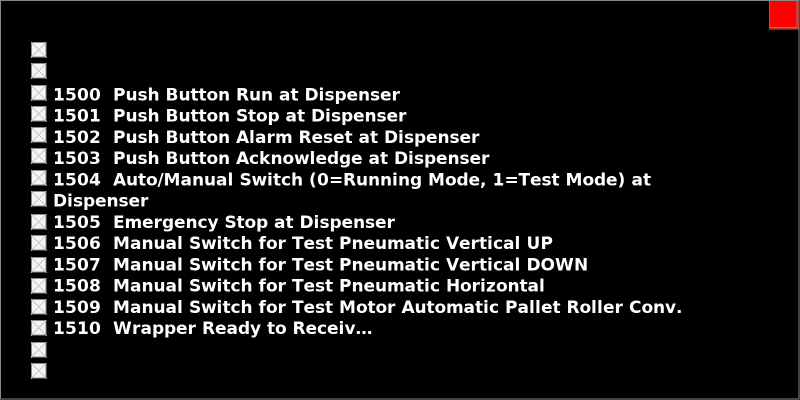
VISUALIZATION P2_DI6  // 800x400, background image 
    ImageSwitcher (31,42 15x15), variable: InputOutput_GVL.Digital_Input[81], behaviour: TOGGLE
    Label (50,16 677x391), "1500 Push Button Run at Dispenser 1501 Push Button Stop at Dispenser 1502 Push Button Alarm Reset at Dispenser 1503 Push Button Acknowledge at Dispenser 1504 Auto/Manual Switch (0=Running Mode, 1=Test Mode) at Dispenser 1505 Emergency Stop at Dispenser 1506 Manual Switch for Test Pneumatic Vertical UP 1507 Manual Switch for Test Pneumatic Vertical DOWN 1508 Manual Switch for Test Pneumatic Horizontal 1509 Manual Switch for Test Motor Automatic Pallet Roller Conv. 1510 Wrapper Ready to Receive 1511 End of Transfer Pallet in Infeed 1512 Pallet Ready in Outfeed 1513 Emergency Stop Wrapper is Active 1514 Status Bypass Wrapper Existing 1515 Pressure Switch for Pallet Dispenser"
    ImageSwitcher (31,63 15x15), variable: InputOutput_GVL.Digital_Input[82], behaviour: TOGGLE
    ImageSwitcher (31,85 15x15), variable: InputOutput_GVL.Digital_Input[83], behaviour: TOGGLE
    ImageSwitcher (31,106 15x15), variable: InputOutput_GVL.Digital_Input[84], behaviour: TOGGLE
    ImageSwitcher (31,127 15x15), variable: InputOutput_GVL.Digital_Input[85], behaviour: TOGGLE
    ImageSwitcher (31,148 15x15), variable: InputOutput_GVL.Digital_Input[86], behaviour: TOGGLE
    ImageSwitcher (31,170 15x15), variable: InputOutput_GVL.Digital_Input[87], behaviour: TOGGLE
    ImageSwitcher (31,191 15x15), variable: InputOutput_GVL.Digital_Input[88], behaviour: TOGGLE
    ImageSwitcher (31,214 15x15), variable: InputOutput_GVL.Digital_Input[89], behaviour: TOGGLE
    ImageSwitcher (31,235 15x15), variable: InputOutput_GVL.Digital_Input[90], behaviour: TOGGLE
    ImageSwitcher (31,257 15x15), variable: InputOutput_GVL.Digital_Input[91], behaviour: TOGGLE
    ImageSwitcher (31,278 15x15), variable: InputOutput_GVL.Digital_Input[92], behaviour: TOGGLE
    ImageSwitcher (31,299 15x15), variable: InputOutput_GVL.Digital_Input[93], behaviour: TOGGLE
    ImageSwitcher (31,320 15x15), variable: InputOutput_GVL.Digital_Input[94], behaviour: TOGGLE
    ImageSwitcher (31,342 15x15), variable: InputOutput_GVL.Digital_Input[95], behaviour: TOGGLE
    ImageSwitcher (31,363 15x15), variable: InputOutput_GVL.Digital_Input[96], behaviour: TOGGLE
    Button (769,-1 30x30), image: VisuSymbols.Symbols.Wrong
        OnMouseClick: CloseDialog Dialog=P2_DI6, Result=OK, NumpadKeypadSet=True
END_VISUALIZATION

(* stored: Version 1.1.0.1, ProductVersion 3.1.4024.12
   Visu P2_DI6: Id {812ca5f8-07a3-4b22-81a6-bbb8bf0908c0} *)
